{attribute addProperty BoxType "EL5152-0000-0016"}
{attribute addProperty Id "Set_counter_doneAT %I*BOOL813Extrapolation_stallAT %I*BOOL818Status_of_input_AAT %I*BOOL819Status_of_input_BAT %I*BOOL8110Sync_errorAT %I*BOOL8132TxPDO_ToggleAT %I*BOOL819Counter_valueAT %I*UINT16217"}
{attribute addProperty CRC "4116829457"}
{attribute addProperty SizeInBites "64"}
{attribute addProperty SizeInBytes "8"}
TYPE ENC_Status_compact_Channel_F561D511 :
STRUCT
	{attribute addProperty Name "Set_counter_done"}
	Set_counter_done AT %I* : BOOL;
	{attribute addProperty Name "Extrapolation_stall"}
	Extrapolation_stall AT %I* : BOOL;
	{attribute addProperty Name "Status_of_input_A"}
	Status_of_input_A AT %I* : BOOL;
	{attribute addProperty Name "Status_of_input_B"}
	Status_of_input_B AT %I* : BOOL;
	{attribute addProperty Name "Sync_error"}
	Sync_error AT %I* : BOOL;
	{attribute addProperty Name "TxPDO_Toggle"}
	TxPDO_Toggle AT %I* : BOOL;
	{attribute addProperty Name "Counter_value"}
	Counter_value AT %I* : UINT;
END_STRUCT
END_TYPE

(* stored: Version 1.2.0.0, ProductVersion 3.1.4024.9
   DUT ENC_Status_compact_Channel_F561D511: Id {8f611333-0fc2-42cc-b25f-1dd05dc2ef30} *)
